# EPICS autosave request: debian/ioc_stats_settings.req
$(IOC):CA_CLNT_CNT.HIGH
$(IOC):CA_CLNT_CNT.HIHI
$(IOC):CA_CONN_CNT.HIGH
$(IOC):CA_CONN_CNT.HIHI
$(IOC):SUSP_TASK_CNT.HIHI
$(IOC):LOAD.HIGH
$(IOC):LOAD.HIHI
$(IOC):FD_FREE.LOLO
$(IOC):FD_FREE.LOW
